ABB RobotStudio station: Entregable3.rspag

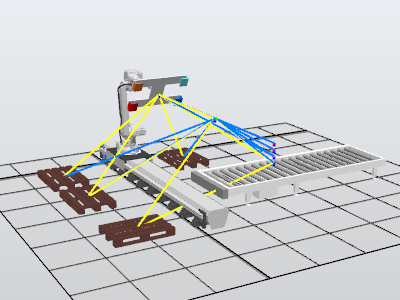
--- station ---
Station Entregable3 (saved by RobotStudio 23.4.10609.1)
Controller Controlador1, task T_ROB1: task frame (RAPID world) sits at (824.5, 292, 460) mm in the station
Controller Controlador1
  mechanical unit TRACK_1: IRBT2005_IRB_STD_INT_0_0_5__01, 1 joints, base frame (0, 0, 0) mm
  mechanical unit ROB_1: IRB4600_20_250_C_01, 6 joints, base frame (0, 0, 0) mm
Layout (positions relative to the parent item):
  - IRBT2005_IRB_STD_INT_0_0_5__01 [mechanism] at (0, 0, 0) mm; joint values [0] (rad or m)
      links: Base, Link1
  - IRB4600_20_250_C_01 [mechanism, from %ABB.RobotStudio.Models.IRB4600%\IRB4600_20_250_C_G_01.rslib] at (824.5, 292, 460) mm; joint values [0, 0, 0, 0, 0.5236, 0] (rad or m)
  - 1200_4000_h2 [part, from %ABB.RobotStudio.Models.Conveyors%\Conveyor 1200 4000 h2.rslib] at (4000, 1000, 0) mm, rotated rx 0 ry 0 rz 90 deg
  - Euro Pallet [graphiccomponentgroup, from Equipment\Euro Pallet.rslib] at (200, -1700, 0) mm
    - Body 1 [part, from Equipment\Euro Pallet.rslib]
  - Euro Pallet_2 [graphiccomponentgroup, from Equipment\Euro Pallet.rslib] at (1700, -1700, 0) mm
    - Body 1 [part, from Equipment\Euro Pallet.rslib]
  - Euro Pallet_3 [graphiccomponentgroup, from Equipment\Euro Pallet.rslib] at (4700, -1700, 0) mm, rotated rx 0 ry 0 rz 90 deg
    - Body 1 [part, from Equipment\Euro Pallet.rslib]
  - Euro Pallet_4 [graphiccomponentgroup, from Equipment\Euro Pallet.rslib] at (200, 1300, 0) mm
    - Body 1 [part, from Equipment\Euro Pallet.rslib]
  - Pinza_para_Pallets [mechanism, from Components\Pinza_para_Pallets.rslib] at (2303.61, 292, 2182.5) mm, rotated rx -180 ry 60 rz -180 deg; joint values [0, 0] (rad or m)
Attachment: IRB4600_20_250_C_01 is attached to IRBT2005_IRB_STD_INT_0_0_5__01 / Link1
Attachment: Pinza_para_Pallets is attached to IRB4600_20_250_C_01 / Link6
EventTableEntry 2433: ActivationMode=2, Cyclic=false, Group=, Trigger=DO_Pinza 2434, Actions=[EventTableActionMechanicalPose 2435, EventTableActionAttach 2436], Comment=
EventTableTriggerIO 2434: Operator=0, IOValue=[1], IRC5Controller=? -1, SignalSource=Controlador1 2457
EventTableActionMechanicalPose 2435: VirtualSignal=, Mechanism=Pinza_para_Pallets 3599, ToPoseName=Cerrada, VirtualSignalValue=[1]
EventTableActionAttach 2436: MountObject=false, FlangeIndext=0, FindNearest=true, AttachmentParent=Pinza_para_Pallets 3599, AttachmentChild=? -1, Offset=[X=1, Y=0, Z=0, W=0, X=0, Y=1, Z=0, W=0, X=0, Y=0, Z=1, W=0, X=0, Y=0, Z=0, W=1]
EventTableTriggerIO 2437: Operator=0, IOValue=[1], IRC5Controller=? -1, SignalSource=Controlador1 2457
EventTableTriggerIO 2438: Operator=0, IOValue=[1], IRC5Controller=? -1, SignalSource=Controlador1 2457
EventTableTriggerIO 2439: Operator=0, IOValue=[1], IRC5Controller=? -1, SignalSource=Controlador1 2457
EventTableTriggerIO 2440: Operator=0, IOValue=[1], IRC5Controller=? -1, SignalSource=Controlador1 2457
EventTableEntry 2444: ActivationMode=2, Cyclic=false, Group=, Trigger=DO_Pinza 3622, Actions=[EventTableActionMechanicalPose 2446, EventTableActionDetach 2447], Comment=
EventTableActionMechanicalPose 2446: VirtualSignal=, Mechanism=Pinza_para_Pallets 3599, ToPoseName=Abierta, VirtualSignalValue=[1]
EventTableActionDetach 2447: AttachmentParent=Pinza_para_Pallets 3599, AttachmentChild=? -1
EventTableTriggerIO 2448: Operator=0, IOValue=[0], IRC5Controller=? -1, SignalSource=Controlador1 2457
EventTableTriggerIO 2449: Operator=0, IOValue=[0], IRC5Controller=? -1, SignalSource=Controlador1 2457
EventTableTriggerIO 2450: Operator=0, IOValue=[0], IRC5Controller=? -1, SignalSource=Controlador1 2457
EventTableTriggerIO 2451: Operator=0, IOValue=[0], IRC5Controller=? -1, SignalSource=Controlador1 2457
EventTableTriggerIO 3621: Operator=0, IOValue=[1], IRC5Controller=? -1, SignalSource=Controlador1 2457
EventTableTriggerIO 3622: Operator=0, IOValue=[0], IRC5Controller=? -1, SignalSource=Controlador1 2457
EventTableTriggerIO 3623: Operator=0, IOValue=[0], IRC5Controller=? -1, SignalSource=Controlador1 2457
EventTableTriggerIO 3657: Operator=0, IOValue=[1], IRC5Controller=? -1, SignalSource=Controlador1 2457
EventTableTriggerIO 3658: Operator=0, IOValue=[1], IRC5Controller=? -1, SignalSource=Controlador1 2457
EventTableTriggerIO 3659: Operator=0, IOValue=[1], IRC5Controller=? -1, SignalSource=Controlador1 2457
EventTableTriggerIO 3660: Operator=0, IOValue=[1], IRC5Controller=? -1, SignalSource=Controlador1 2457
EventTableTriggerIO 3661: Operator=0, IOValue=[1], IRC5Controller=? -1, SignalSource=Controlador1 2457
EventTableTriggerIO 3662: Operator=0, IOValue=[1], IRC5Controller=? -1, SignalSource=Controlador1 2457
EventTableTriggerIO 3663: Operator=0, IOValue=[1], IRC5Controller=? -1, SignalSource=Controlador1 2457
EventTableTriggerIO 3664: Operator=0, IOValue=[1], IRC5Controller=? -1, SignalSource=Controlador1 2457
EventTableTriggerIO 3665: Operator=0, IOValue=[1], IRC5Controller=? -1, SignalSource=Controlador1 2457
EventTableTriggerIO 3666: Operator=0, IOValue=[1], IRC5Controller=? -1, SignalSource=Controlador1 2457
EventTableTriggerIO 3667: Operator=0, IOValue=[1], IRC5Controller=? -1, SignalSource=Controlador1 2457
EventTableTriggerIO 3668: Operator=0, IOValue=[1], IRC5Controller=? -1, SignalSource=Controlador1 2457
EventTableTriggerIO 3669: Operator=0, IOValue=[1], IRC5Controller=? -1, SignalSource=Controlador1 2457
EventTableTriggerIO 3670: Operator=0, IOValue=[1], IRC5Controller=? -1, SignalSource=Controlador1 2457
EventTableTriggerIO 3671: Operator=0, IOValue=[0], IRC5Controller=? -1, SignalSource=Controlador1 2457
EventTableTriggerIO 3672: Operator=0, IOValue=[0], IRC5Controller=? -1, SignalSource=Controlador1 2457
EventTableTriggerIO 3673: Operator=0, IOValue=[0], IRC5Controller=? -1, SignalSource=Controlador1 2457
EventTableTriggerIO 3674: Operator=0, IOValue=[0], IRC5Controller=? -1, SignalSource=Controlador1 2457
EventTableTriggerIO 3675: Operator=0, IOValue=[0], IRC5Controller=? -1, SignalSource=Controlador1 2457
EventTableTriggerIO 3676: Operator=0, IOValue=[0], IRC5Controller=? -1, SignalSource=Controlador1 2457
EventTableTriggerIO 3677: Operator=0, IOValue=[0], IRC5Controller=? -1, SignalSource=Controlador1 2457
EventTableTriggerIO 3678: Operator=0, IOValue=[0], IRC5Controller=? -1, SignalSource=Controlador1 2457
EventTableTriggerIO 3679: Operator=0, IOValue=[0], IRC5Controller=? -1, SignalSource=Controlador1 2457
EventTableTriggerIO 3680: Operator=0, IOValue=[0], IRC5Controller=? -1, SignalSource=Controlador1 2457
EventTableTriggerIO 3681: Operator=0, IOValue=[0], IRC5Controller=? -1, SignalSource=Controlador1 2457
EventTableTriggerIO 3682: Operator=0, IOValue=[0], IRC5Controller=? -1, SignalSource=Controlador1 2457
EventTableTriggerIO 3683: Operator=0, IOValue=[0], IRC5Controller=? -1, SignalSource=Controlador1 2457
EventTableTriggerIO 3684: Operator=0, IOValue=[0], IRC5Controller=? -1, SignalSource=Controlador1 2457
EventTableTriggerIO 3980: Operator=0, IOValue=[1], IRC5Controller=? -1, SignalSource=Controlador1 2457
EventTableTriggerIO 3981: Operator=0, IOValue=[1], IRC5Controller=? -1, SignalSource=Controlador1 2457
EventTableTriggerIO 3982: Operator=0, IOValue=[1], IRC5Controller=? -1, SignalSource=Controlador1 2457
EventTableTriggerIO 3983: Operator=0, IOValue=[1], IRC5Controller=? -1, SignalSource=Controlador1 2457
EventTableTriggerIO 3984: Operator=0, IOValue=[1], IRC5Controller=? -1, SignalSource=Controlador1 2457
EventTableTriggerIO 3985: Operator=0, IOValue=[1], IRC5Controller=? -1, SignalSource=Controlador1 2457
EventTableTriggerIO 3986: Operator=0, IOValue=[1], IRC5Controller=? -1, SignalSource=Controlador1 2457
EventTableTriggerIO 3987: Operator=0, IOValue=[0], IRC5Controller=? -1, SignalSource=Controlador1 2457
EventTableTriggerIO 3988: Operator=0, IOValue=[0], IRC5Controller=? -1, SignalSource=Controlador1 2457
EventTableTriggerIO 3989: Operator=0, IOValue=[0], IRC5Controller=? -1, SignalSource=Controlador1 2457
EventTableTriggerIO 3990: Operator=0, IOValue=[0], IRC5Controller=? -1, SignalSource=Controlador1 2457
EventTableTriggerIO 3991: Operator=0, IOValue=[0], IRC5Controller=? -1, SignalSource=Controlador1 2457
EventTableTriggerIO 3992: Operator=0, IOValue=[0], IRC5Controller=? -1, SignalSource=Controlador1 2457
EventTableTriggerIO 3993: Operator=0, IOValue=[0], IRC5Controller=? -1, SignalSource=Controlador1 2457
EventTableEntry 3994: ActivationMode=2, Cyclic=false, Group=, Trigger=DO_Cinta 3995, Actions=[EventTableActionMechanicalPose 3996], Comment=
EventTableTriggerIO 3995: Operator=0, IOValue=[1], IRC5Controller=? -1, SignalSource=Controlador1 2457
EventTableActionMechanicalPose 3996: VirtualSignal=, Mechanism=IRBT2005_IRB_STD_INT_0_0_5__01 2366, ToPoseName=Descarga, VirtualSignalValue=[1]
EventTableTriggerIO 3997: Operator=0, IOValue=[1], IRC5Controller=? -1, SignalSource=Controlador1 2457
EventTableTriggerIO 3998: Operator=0, IOValue=[1], IRC5Controller=? -1, SignalSource=Controlador1 2457
EventTableTriggerIO 3999: Operator=0, IOValue=[1], IRC5Controller=? -1, SignalSource=Controlador1 2457
EventTableTriggerIO 4000: Operator=0, IOValue=[1], IRC5Controller=? -1, SignalSource=Controlador1 2457
EventTableTriggerIO 4001: Operator=0, IOValue=[1], IRC5Controller=? -1, SignalSource=Controlador1 2457
EventTableEntry 4002: ActivationMode=2, Cyclic=false, Group=, Trigger=DO_Cinta 4003, Actions=[EventTableActionMechanicalPose 4004], Comment=
EventTableTriggerIO 4003: Operator=0, IOValue=[0], IRC5Controller=? -1, SignalSource=Controlador1 2457
EventTableActionMechanicalPose 4004: VirtualSignal=, Mechanism=IRBT2005_IRB_STD_INT_0_0_5__01 2366, ToPoseName=Home, VirtualSignalValue=[1]
EventTableTriggerIO 4005: Operator=0, IOValue=[0], IRC5Controller=? -1, SignalSource=Controlador1 2457
EventTableTriggerIO 4006: Operator=0, IOValue=[0], IRC5Controller=? -1, SignalSource=Controlador1 2457
EventTableTriggerIO 4007: Operator=0, IOValue=[0], IRC5Controller=? -1, SignalSource=Controlador1 2457
EventTableTriggerIO 4008: Operator=0, IOValue=[0], IRC5Controller=? -1, SignalSource=Controlador1 2457
EventTableTriggerIO 4009: Operator=0, IOValue=[0], IRC5Controller=? -1, SignalSource=Controlador1 2457
EventTableTriggerIO 4070: Operator=0, IOValue=[1], IRC5Controller=? -1, SignalSource=Controlador1 2457
EventTableTriggerIO 4071: Operator=0, IOValue=[1], IRC5Controller=? -1, SignalSource=Controlador1 2457
EventTableTriggerIO 4072: Operator=0, IOValue=[1], IRC5Controller=? -1, SignalSource=Controlador1 2457
EventTableTriggerIO 4073: Operator=0, IOValue=[1], IRC5Controller=? -1, SignalSource=Controlador1 2457
EventTableTriggerIO 4074: Operator=0, IOValue=[1], IRC5Controller=? -1, SignalSource=Controlador1 2457
EventTableTriggerIO 4075: Operator=0, IOValue=[1], IRC5Controller=? -1, SignalSource=Controlador1 2457
EventTableTriggerIO 4076: Operator=0, IOValue=[1], IRC5Controller=? -1, SignalSource=Controlador1 2457
EventTableTriggerIO 4077: Operator=0, IOValue=[1], IRC5Controller=? -1, SignalSource=Controlador1 2457
EventTableTriggerIO 4078: Operator=0, IOValue=[1], IRC5Controller=? -1, SignalSource=Controlador1 2457
EventTableTriggerIO 4079: Operator=0, IOValue=[1], IRC5Controller=? -1, SignalSource=Controlador1 2457
EventTableTriggerIO 4080: Operator=0, IOValue=[1], IRC5Controller=? -1, SignalSource=Controlador1 2457
EventTableTriggerIO 4081: Operator=0, IOValue=[1], IRC5Controller=? -1, SignalSource=Controlador1 2457
EventTableTriggerIO 4082: Operator=0, IOValue=[1], IRC5Controller=? -1, SignalSource=Controlador1 2457
EventTableTriggerIO 4083: Operator=0, IOValue=[1], IRC5Controller=? -1, SignalSource=Controlador1 2457
EventTableTriggerIO 4084: Operator=0, IOValue=[1], IRC5Controller=? -1, SignalSource=Controlador1 2457
EventTableTriggerIO 4085: Operator=0, IOValue=[1], IRC5Controller=? -1, SignalSource=Controlador1 2457
EventTableTriggerIO 4086: Operator=0, IOValue=[1], IRC5Controller=? -1, SignalSource=Controlador1 2457
EventTableTriggerIO 4087: Operator=0, IOValue=[0], IRC5Controller=? -1, SignalSource=Controlador1 2457
EventTableTriggerIO 4088: Operator=0, IOValue=[0], IRC5Controller=? -1, SignalSource=Controlador1 2457
EventTableTriggerIO 4089: Operator=0, IOValue=[0], IRC5Controller=? -1, SignalSource=Controlador1 2457
EventTableTriggerIO 4090: Operator=0, IOValue=[0], IRC5Controller=? -1, SignalSource=Controlador1 2457
EventTableTriggerIO 4091: Operator=0, IOValue=[0], IRC5Controller=? -1, SignalSource=Controlador1 2457
EventTableTriggerIO 4092: Operator=0, IOValue=[0], IRC5Controller=? -1, SignalSource=Controlador1 2457
EventTableTriggerIO 4093: Operator=0, IOValue=[0], IRC5Controller=? -1, SignalSource=Controlador1 2457
EventTableTriggerIO 4094: Operator=0, IOValue=[0], IRC5Controller=? -1, SignalSource=Controlador1 2457
EventTableTriggerIO 4095: Operator=0, IOValue=[0], IRC5Controller=? -1, SignalSource=Controlador1 2457
EventTableTriggerIO 4096: Operator=0, IOValue=[0], IRC5Controller=? -1, SignalSource=Controlador1 2457
EventTableTriggerIO 4097: Operator=0, IOValue=[0], IRC5Controller=? -1, SignalSource=Controlador1 2457
EventTableTriggerIO 4098: Operator=0, IOValue=[0], IRC5Controller=? -1, SignalSource=Controlador1 2457
EventTableTriggerIO 4099: Operator=0, IOValue=[0], IRC5Controller=? -1, SignalSource=Controlador1 2457
EventTableTriggerIO 4100: Operator=0, IOValue=[0], IRC5Controller=? -1, SignalSource=Controlador1 2457
EventTableTriggerIO 4101: Operator=0, IOValue=[0], IRC5Controller=? -1, SignalSource=Controlador1 2457
EventTableTriggerIO 4102: Operator=0, IOValue=[0], IRC5Controller=? -1, SignalSource=Controlador1 2457
EventTableTriggerIO 4103: Operator=0, IOValue=[0], IRC5Controller=? -1, SignalSource=Controlador1 2457
EventTableTriggerIO 4104: Operator=0, IOValue=[1], IRC5Controller=? -1, SignalSource=Controlador1 2457
EventTableTriggerIO 4105: Operator=0, IOValue=[1], IRC5Controller=? -1, SignalSource=Controlador1 2457
EventTableTriggerIO 4106: Operator=0, IOValue=[1], IRC5Controller=? -1, SignalSource=Controlador1 2457
EventTableTriggerIO 4107: Operator=0, IOValue=[1], IRC5Controller=? -1, SignalSource=Controlador1 2457
EventTableTriggerIO 4108: Operator=0, IOValue=[1], IRC5Controller=? -1, SignalSource=Controlador1 2457
EventTableTriggerIO 4109: Operator=0, IOValue=[1], IRC5Controller=? -1, SignalSource=Controlador1 2457
EventTableTriggerIO 4110: Operator=0, IOValue=[1], IRC5Controller=? -1, SignalSource=Controlador1 2457
EventTableTriggerIO 4111: Operator=0, IOValue=[1], IRC5Controller=? -1, SignalSource=Controlador1 2457
EventTableTriggerIO 4112: Operator=0, IOValue=[1], IRC5Controller=? -1, SignalSource=Controlador1 2457
EventTableTriggerIO 4113: Operator=0, IOValue=[1], IRC5Controller=? -1, SignalSource=Controlador1 2457
EventTableTriggerIO 4114: Operator=0, IOValue=[1], IRC5Controller=? -1, SignalSource=Controlador1 2457
EventTableTriggerIO 4115: Operator=0, IOValue=[1], IRC5Controller=? -1, SignalSource=Controlador1 2457
EventTableTriggerIO 4116: Operator=0, IOValue=[1], IRC5Controller=? -1, SignalSource=Controlador1 2457
EventTableTriggerIO 4117: Operator=0, IOValue=[1], IRC5Controller=? -1, SignalSource=Controlador1 2457
EventTableTriggerIO 4118: Operator=0, IOValue=[1], IRC5Controller=? -1, SignalSource=Controlador1 2457
EventTableTriggerIO 4119: Operator=0, IOValue=[1], IRC5Controller=? -1, SignalSource=Controlador1 2457
EventTableTriggerIO 4120: Operator=0, IOValue=[1], IRC5Controller=? -1, SignalSource=Controlador1 2457
EventTableTriggerIO 4121: Operator=0, IOValue=[0], IRC5Controller=? -1, SignalSource=Controlador1 2457
EventTableTriggerIO 4122: Operator=0, IOValue=[0], IRC5Controller=? -1, SignalSource=Controlador1 2457
EventTableTriggerIO 4123: Operator=0, IOValue=[0], IRC5Controller=? -1, SignalSource=Controlador1 2457
EventTableTriggerIO 4124: Operator=0, IOValue=[0], IRC5Controller=? -1, SignalSource=Controlador1 2457
EventTableTriggerIO 4125: Operator=0, IOValue=[0], IRC5Controller=? -1, SignalSource=Controlador1 2457
EventTableTriggerIO 4126: Operator=0, IOValue=[0], IRC5Controller=? -1, SignalSource=Controlador1 2457
EventTableTriggerIO 4127: Operator=0, IOValue=[0], IRC5Controller=? -1, SignalSource=Controlador1 2457
EventTableTriggerIO 4128: Operator=0, IOValue=[0], IRC5Controller=? -1, SignalSource=Controlador1 2457
EventTableTriggerIO 4129: Operator=0, IOValue=[0], IRC5Controller=? -1, SignalSource=Controlador1 2457
EventTableTriggerIO 4130: Operator=0, IOValue=[0], IRC5Controller=? -1, SignalSource=Controlador1 2457
EventTableTriggerIO 4131: Operator=0, IOValue=[0], IRC5Controller=? -1, SignalSource=Controlador1 2457
EventTableTriggerIO 4132: Operator=0, IOValue=[0], IRC5Controller=? -1, SignalSource=Controlador1 2457
EventTableTriggerIO 4133: Operator=0, IOValue=[0], IRC5Controller=? -1, SignalSource=Controlador1 2457
EventTableTriggerIO 4134: Operator=0, IOValue=[0], IRC5Controller=? -1, SignalSource=Controlador1 2457
EventTableTriggerIO 4135: Operator=0, IOValue=[0], IRC5Controller=? -1, SignalSource=Controlador1 2457
EventTableTriggerIO 4136: Operator=0, IOValue=[0], IRC5Controller=? -1, SignalSource=Controlador1 2457
EventTableTriggerIO 4137: Operator=0, IOValue=[0], IRC5Controller=? -1, SignalSource=Controlador1 2457
EventTableTriggerIO 4251: Operator=0, IOValue=[1], IRC5Controller=? -1, SignalSource=Controlador1 2457
EventTableTriggerIO 4252: Operator=0, IOValue=[1], IRC5Controller=? -1, SignalSource=Controlador1 2457
EventTableTriggerIO 4253: Operator=0, IOValue=[1], IRC5Controller=? -1, SignalSource=Controlador1 2457
EventTableTriggerIO 4254: Operator=0, IOValue=[1], IRC5Controller=? -1, SignalSource=Controlador1 2457
EventTableTriggerIO 4255: Operator=0, IOValue=[1], IRC5Controller=? -1, SignalSource=Controlador1 2457
EventTableTriggerIO 4256: Operator=0, IOValue=[1], IRC5Controller=? -1, SignalSource=Controlador1 2457
EventTableTriggerIO 4257: Operator=0, IOValue=[1], IRC5Controller=? -1, SignalSource=Controlador1 2457
EventTableTriggerIO 4258: Operator=0, IOValue=[1], IRC5Controller=? -1, SignalSource=Controlador1 2457
EventTableTriggerIO 4259: Operator=0, IOValue=[1], IRC5Controller=? -1, SignalSource=Controlador1 2457
EventTableTriggerIO 4260: Operator=0, IOValue=[0], IRC5Controller=? -1, SignalSource=Controlador1 2457
EventTableTriggerIO 4261: Operator=0, IOValue=[0], IRC5Controller=? -1, SignalSource=Controlador1 2457
EventTableTriggerIO 4262: Operator=0, IOValue=[0], IRC5Controller=? -1, SignalSource=Controlador1 2457
EventTableTriggerIO 4263: Operator=0, IOValue=[0], IRC5Controller=? -1, SignalSource=Controlador1 2457
EventTableTriggerIO 4264: Operator=0, IOValue=[0], IRC5Controller=? -1, SignalSource=Controlador1 2457
EventTableTriggerIO 4265: Operator=0, IOValue=[0], IRC5Controller=? -1, SignalSource=Controlador1 2457
EventTableTriggerIO 4266: Operator=0, IOValue=[0], IRC5Controller=? -1, SignalSource=Controlador1 2457
EventTableTriggerIO 4267: Operator=0, IOValue=[0], IRC5Controller=? -1, SignalSource=Controlador1 2457
EventTableTriggerIO 4268: Operator=0, IOValue=[0], IRC5Controller=? -1, SignalSource=Controlador1 2457
EventTableTriggerIO 4269: Operator=0, IOValue=[1], IRC5Controller=? -1, SignalSource=Controlador1 2457
EventTableTriggerIO 4270: Operator=0, IOValue=[1], IRC5Controller=? -1, SignalSource=Controlador1 2457
EventTableTriggerIO 4271: Operator=0, IOValue=[1], IRC5Controller=? -1, SignalSource=Controlador1 2457
EventTableTriggerIO 4272: Operator=0, IOValue=[1], IRC5Controller=? -1, SignalSource=Controlador1 2457
EventTableTriggerIO 4273: Operator=0, IOValue=[1], IRC5Controller=? -1, SignalSource=Controlador1 2457
EventTableTriggerIO 4274: Operator=0, IOValue=[1], IRC5Controller=? -1, SignalSource=Controlador1 2457
EventTableTriggerIO 4275: Operator=0, IOValue=[1], IRC5Controller=? -1, SignalSource=Controlador1 2457
EventTableTriggerIO 4276: Operator=0, IOValue=[1], IRC5Controller=? -1, SignalSource=Controlador1 2457
EventTableTriggerIO 4277: Operator=0, IOValue=[1], IRC5Controller=? -1, SignalSource=Controlador1 2457
EventTableTriggerIO 4278: Operator=0, IOValue=[0], IRC5Controller=? -1, SignalSource=Controlador1 2457
EventTableTriggerIO 4279: Operator=0, IOValue=[0], IRC5Controller=? -1, SignalSource=Controlador1 2457
EventTableTriggerIO 4280: Operator=0, IOValue=[0], IRC5Controller=? -1, SignalSource=Controlador1 2457
EventTableTriggerIO 4281: Operator=0, IOValue=[0], IRC5Controller=? -1, SignalSource=Controlador1 2457
EventTableTriggerIO 4282: Operator=0, IOValue=[0], IRC5Controller=? -1, SignalSource=Controlador1 2457
EventTableTriggerIO 4283: Operator=0, IOValue=[0], IRC5Controller=? -1, SignalSource=Controlador1 2457
EventTableTriggerIO 4284: Operator=0, IOValue=[0], IRC5Controller=? -1, SignalSource=Controlador1 2457
EventTableTriggerIO 4285: Operator=0, IOValue=[0], IRC5Controller=? -1, SignalSource=Controlador1 2457
EventTableTriggerIO 4286: Operator=0, IOValue=[0], IRC5Controller=? -1, SignalSource=Controlador1 2457
Targets, tools, work objects and paths stored in the station and not in the controller backup, written as RAPID:
! task T_ROB1
MODULE CalibData
  PERS tooldata Pinza_para_Pallets_1:=[TRUE,[[0,0,160],[1,0,0,0]],[5,[0,0,80],[1,0,0,0],0,0,0]];
ENDMODULE

! task T_ROB1
MODULE Module1
  CONST robtarget Home:=[[1617.676223927,0,1642.5],[0,0,1,0],[0,0,0,0],[0,9E+09,9E+09,9E+09,9E+09,9E+09]];
  CONST robtarget Pallet_1:=[[-6.53,-1592.857,-355.998],[0,0,1,0],[-2,0,0,0],[0,9E+09,9E+09,9E+09,9E+09,9E+09]];
  CONST robtarget Pallet_2:=[[1466.445,-1582.941,-356.002],[0,1,0,0],[-1,0,1,0],[0,9E+09,9E+09,9E+09,9E+09,9E+09]];
  CONST robtarget Pallet_3:=[[-41.934,1427.208,-355.998],[0,0,1,0],[0,0,0,0],[0,9E+09,9E+09,9E+09,9E+09,9E+09]];
  CONST robtarget Cinta:=[[2534.438,2270.837,84.535],[0,-0.707106781,0.707106781,0],[0,0,0,0],[2281.316725979,9E+09,9E+09,9E+09,9E+09,9E+09]];
  CONST robtarget Download:=[[3898.992949906,0,1642.5],[0,0,1,0],[0,0,0,0],[2281.316725979,9E+09,9E+09,9E+09,9E+09,9E+09]];
  CONST robtarget Cinta_2:=[[2534.438,2270.837,230.535],[0,-0.707106781,0.707106781,0],[0,0,0,0],[2281.316725979,9E+09,9E+09,9E+09,9E+09,9E+09]];
  CONST robtarget Cinta_3:=[[2534.438,2270.837,376.535],[0,-0.707106781,0.707106781,0],[0,0,-1,0],[2281.316725979,9E+09,9E+09,9E+09,9E+09,9E+09]];
  CONST robtarget Cinta_4:=[[2534.438,2270.837,522.535],[0,-0.707106781,0.707106781,0],[0,0,-1,0],[2281.316725979,9E+09,9E+09,9E+09,9E+09,9E+09]];
  CONST robtarget Pallet_4:=[[3464.692,-1392.703,-355.996],[0,0.707106781,0.707106781,0],[-1,0,0,0],[2281.316725979,9E+09,9E+09,9E+09,9E+09,9E+09]];
  PROC Pallet2()
    MoveL Home,v1000,fine,Pinza_para_Pallets_1\WObj:=wobj0;
    MoveL Pallet_2,v1000,fine,Pinza_para_Pallets_1\WObj:=wobj0;
    SetDO DO_Pinza,1;
    WaitTime 2;
    MoveL Download,v1000,z100,Pinza_para_Pallets_1\WObj:=wobj0;
    MoveL Cinta,v1000,fine,Pinza_para_Pallets_1\WObj:=wobj0;
    SetDO DO_Pinza,0;
    WaitTime 2;
    MoveL Home,v1000,fine,Pinza_para_Pallets_1\WObj:=wobj0;
  ENDPROC
  PROC Pallet1()
    MoveL Home,v1000,z100,Pinza_para_Pallets_1\WObj:=wobj0;
    MoveL Pallet_1,v1000,fine,Pinza_para_Pallets_1\WObj:=wobj0;
    SetDO DO_Pinza,1;
    WaitTime 2;
    MoveL Home,v1000,fine,Pinza_para_Pallets_1\WObj:=wobj0;
    MoveL Pallet_1,v1000,fine,Pinza_para_Pallets_1\WObj:=wobj0;
    SetDO DO_Pinza,0;
    WaitTime 2;
    MoveL Home,v1000,fine,Pinza_para_Pallets_1\WObj:=wobj0;
  ENDPROC
  PROC Pallet3()
    MoveL Home,v1000,z100,Pinza_para_Pallets_1\WObj:=wobj0;
    MoveL Pallet_3,v1000,fine,Pinza_para_Pallets_1\WObj:=wobj0;
    SetDO DO_Pinza,1;
    WaitTime 2;
    MoveL Home,v1000,fine,Pinza_para_Pallets_1\WObj:=wobj0;
    MoveL Pallet_3,v1000,fine,Pinza_para_Pallets_1\WObj:=wobj0;
    SetDO DO_Pinza,0;
    WaitTime 2;
    MoveL Home,v1000,fine,Pinza_para_Pallets_1\WObj:=wobj0;
  ENDPROC
  PROC Pallet4()
    MoveL Home,v1000,fine,Pinza_para_Pallets_1\WObj:=wobj0;
    MoveL Download,v1000,z100,Pinza_para_Pallets_1\WObj:=wobj0;
    MoveL Pallet_4,v1000,fine,Pinza_para_Pallets_1\WObj:=wobj0;
    SetDO DO_Pinza,1;
    WaitTime 2;
    MoveL Cinta,v1000,z100,Pinza_para_Pallets_1\WObj:=wobj0;
    SetDO DO_Pinza,0;
    WaitTime 2;
    MoveL Home,v1000,fine,Pinza_para_Pallets_1\WObj:=wobj0;
  ENDPROC
  PROC Final()
    MoveL Home,v1000,fine,Pinza_para_Pallets_1\WObj:=wobj0;
    MoveL Pallet_1,v1000,fine,Pinza_para_Pallets_1\WObj:=wobj0;
    SetDO DO_Pinza,1;
    WaitTime 2;
    MoveL Download,v1000,fine,Pinza_para_Pallets_1\WObj:=wobj0;
    MoveL Cinta,v1000,fine,Pinza_para_Pallets_1\WObj:=wobj0;
    SetDO DO_Pinza,0;
    MoveL Home,v1000,fine,Pinza_para_Pallets_1\WObj:=wobj0;
    MoveL Pallet_2,v1000,fine,Pinza_para_Pallets_1\WObj:=wobj0;
    SetDO DO_Pinza,1;
    WaitTime 2;
    MoveL Download,v1000,fine,Pinza_para_Pallets_1\WObj:=wobj0;
    MoveL Cinta_2,v1000,fine,Pinza_para_Pallets_1\WObj:=wobj0;
    SetDO DO_Pinza,0;
    MoveL Home,v1000,fine,Pinza_para_Pallets_1\WObj:=wobj0;
    MoveL Pallet_3,v1000,fine,Pinza_para_Pallets_1\WObj:=wobj0;
    SetDO DO_Pinza,1;
    WaitTime 2;
    MoveL Download,v1000,fine,Pinza_para_Pallets_1\WObj:=wobj0;
    MoveL Cinta_3,v1000,fine,Pinza_para_Pallets_1\WObj:=wobj0;
    SetDO DO_Pinza,0;
    MoveL Download,v1000,fine,Pinza_para_Pallets_1\WObj:=wobj0;
    MoveL Pallet_4,v1000,fine,Pinza_para_Pallets_1\WObj:=wobj0;
    SetDO DO_Pinza,1;
    WaitTime 2;
    MoveL Download,v1000,fine,Pinza_para_Pallets_1\WObj:=wobj0;
    MoveL Cinta_4,v1000,fine,Pinza_para_Pallets_1\WObj:=wobj0;
    SetDO DO_Pinza,0;
    MoveL Home,v1000,fine,Pinza_para_Pallets_1\WObj:=wobj0;
  ENDPROC
ENDMODULE


--- Controller Data/Controlador1/RAPID/TASK1/PROGMOD/Module1.mod ---
MODULE Module1
    !***********************************************************
    !
    ! M?dulo:  Module1
    !
    ! Descripción:
    !   <Introduzca la descripción aquí>
    !
    ! Autor: Javier
    !
    ! Versión: 1.0
    !
    !***********************************************************


    !***********************************************************
    !
    ! Procedimiento Main
    !
    !   Este es el punto de entrada de su programa
    !
    !***********************************************************
    PROC main()
        !Add your code here
    ENDPROC
ENDMODULE

--- Controller Data/Controlador1/SYSPAR/EIO.cfg ---
EIO:CFG_1.0:6:1::
#
EIO_SIGNAL:

      -Name "DO_Pinza" -SignalType "DO" -Access "All"

      -Name "DO_Cinta" -SignalType "DO" -Access "All"
